Universal Robots PolyScope program: TEST_THREAD.urp

Program TEST_THREAD (installation=GD directory=/programs/GD createdIn=5.13.0 lastSavedIn=5.13.0 robotSerialNumber=20235201009)
Calibrated DH parameters: a=[0.000068, -0.459527, -0.565386, -0.00004, -0.000074, 0]; d=[0.180653, 1135.485256, -1146.280412, 10.969393, 0.119732, 0.115458]; alpha=[1.570272, -0.000356, 0.007489, 1.569439, -1.570428, 0]; deltaTheta=[0, -0.72179, 6.862965, 0.14202, 0, 0]
InitVariablesNode
BeforeStart
  Script file /programs/GD/THREAD/THREAD_TEST.script
    | thread THREAD_TEST():
    |   THREAD_TEST_FLAG=0
    |   var_2=0
    |   while (var_2<10):
    |     sleep(1.0)
    |     var_2=var_2+1
    |   end
    |   THREAD_TEST_FLAG=1
    | end
    | def RUN_THREAD_TEST():
    |   return run THREAD_TEST()
    | end
    | def JOIN_THREAD_TEST(thrd):
    |   join thrd
    | end
  Script file /programs/GD/THREAD/THREAD_ROVI.script
    | thread THREAD_ROVI():
    |   THREAD_ROVI_FLAG=0
    |   if ((not ROVI_RECIPE(read_input_integer_register(2)+WorkNoOffset))):
    |     global SubPrgResult=rovi_err
    |     sleep(999999.0)
    |   end
    |   if ((not ROVI_RESET())):
    |     global SubPrgResult=rovi_err
    |     sleep(999999.0)
    |   end
    |   if ((  not  ROVI_CAPTURE())):
    |     global SubPrgResult=rovi_err
    |     sleep(999999.0)
    |   end
    |   global Y2=ROVI_SOLVE()
    |   if ((Y2[0] == 10000.)):
    |     global SubPrgResult=rovi_err
    |     sleep(999999.0)
    |   end
    |   THREAD_ROVI_FLAG=1
    | end
    | def RUN_THREAD_ROVI():
    |   return run THREAD_ROVI()
    | end
    | def JOIN_THREAD_ROVI(thrd):
    |   join thrd
    | end
    | def RESET_THREAD_ROVI():
    |   THREAD_ROVI_FLAG=2
    | end
    | def KILL_THREAD_ROVI(thrd):
    |   if (THREAD_ROVI_FLAG==0):
    |     kill thrd
    |   end
    | end
Robot Program (runOnlyOnce=true)
  test_mode := 1
  MoveJ speed 60 deg/s, acceleration 80 deg/s^2 (useActiveTCP=true) feature=Base
    Waypoint ウェイポイント_1: TCP in base x=-3.296 y=-333.288 z=195.515 mm, rx=-0.0179 ry=-3.1401 rz=0.0062 rad; joints [-66.158, -59.903, -118.155, -91.793, 90.282, 24.485] deg; TCP offset x=0 y=90 z=420 mm, rx=0 ry=0 rz=0 rad
  var_1 := 0
  var_2 := 0
  If test_mode≟0
    Folder SINGLE
      Loop While (checkContinuously=false) expression=var_1<10
        Wait Sleep waitTime=1
        var_1 := var_1+1
      Popup Message (haltProgram=false message='SINGLE' done! inputType=Text)
      MoveL speed 250 mm/s, acceleration 1200 mm/s^2 (useActiveTCP=true) feature=Base
        Waypoint ウェイポイント_2: TCP in base x=-3.267 y=-780.038 z=195.535 mm, rx=-0.018 ry=-3.1401 rz=0.0063 rad; joints [-78.704, -105.216, -78.971, -85.627, 90.306, 11.98] deg
      Wait Sleep waitTime=0.5
      MoveL speed 250 mm/s, acceleration 1200 mm/s^2 (useActiveTCP=true) feature=Base
        Waypoint ウェイポイント_1: TCP in base x=-3.296 y=-333.288 z=195.515 mm, rx=-0.0179 ry=-3.1401 rz=0.0062 rad; joints [-66.158, -59.903, -118.155, -91.793, 90.282, 24.485] deg
  ElseIf test_mode≟1
    Folder THREAD
      thrd := RUN_THREAD_TEST()
      MoveL speed 250 mm/s, acceleration 1200 mm/s^2 (useActiveTCP=true) feature=Base
        Waypoint ウェイポイント_2: TCP in base x=-3.267 y=-780.038 z=195.535 mm, rx=-0.018 ry=-3.1401 rz=0.0063 rad; joints [-78.704, -105.216, -78.971, -85.627, 90.306, 11.98] deg
      Wait Sleep waitTime=0.5
      Script: JOIN_THREAD_TEST(thrd)
      Popup Message (haltProgram=false message='THREAD' done! inputType=Text)
      MoveL speed 250 mm/s, acceleration 1200 mm/s^2 (useActiveTCP=true) feature=Base
        Waypoint ウェイポイント_1: TCP in base x=-3.296 y=-333.288 z=195.515 mm, rx=-0.0179 ry=-3.1401 rz=0.0062 rad; joints [-66.158, -59.903, -118.155, -91.793, 90.282, 24.485] deg
  ElseIf test_mode≟2
    Folder THREAD
      thrd := RUN_THREAD_ROVI()
      MoveL speed 250 mm/s, acceleration 1200 mm/s^2 (useActiveTCP=true) feature=Base
        Waypoint ウェイポイント_2: TCP in base x=-3.267 y=-780.038 z=195.535 mm, rx=-0.018 ry=-3.1401 rz=0.0063 rad; joints [-78.704, -105.216, -78.971, -85.627, 90.306, 11.98] deg
      Wait Sleep waitTime=0.5
      Script: JOIN_THREAD_ROVI(thrd)
      Popup Message (haltProgram=false message='THREAD' done! inputType=Text)
      MoveL speed 250 mm/s, acceleration 1200 mm/s^2 (useActiveTCP=true) feature=Base
        Waypoint ウェイポイント_1: TCP in base x=-3.296 y=-333.288 z=195.515 mm, rx=-0.0179 ry=-3.1401 rz=0.0062 rad; joints [-66.158, -59.903, -118.155, -91.793, 90.282, 24.485] deg
